FUNCTION RFID_Sensor_Detect : RFID_Sensor_Errors
VAR_INPUT
	Sensor :  REFERENCE TO RFID_Sensor;
END_VAR

VAR_IN_OUT
	Q : BOOL;
END_VAR

VAR
END_VAR

IF Sensor.IN_Not_Connected_To_Read_Write_Head THEN
	RFID_Sensor_Detect := RFID_Sensor_Errors.Not_Connected;
	Q := FALSE;
ELSIF Sensor.IN_Antenna_Detuned_AT_HF_Read_Write_Head THEN
	RFID_Sensor_Detect := RFID_Sensor_Errors.Antenna_Detuned;
	Q := FALSE;
ELSE
	RFID_Sensor_Detect := RFID_Sensor_Errors.None;
	Q := Sensor.IN_Tag_Presant_At_R_W_Head;
END_IF

END_FUNCTION

(* stored: Version 1.1.0.1, ProductVersion 3.1.4024.10
   POU RFID_Sensor_Detect: Id {3809c1b7-b592-4b3f-89ec-357b213f79ca}, SpecialFunc None *)
